FUNCTION_BLOCK PI (* PI FB *)
  (* Standard: 61499-2 *)
  (* Version 1.0, 2026-04-19, Thomas Mayr *)
  PACKAGE eclipse4diac::controlengineering;
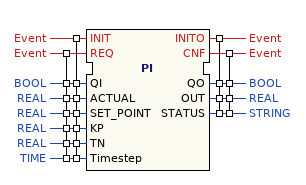
  EVENT_INPUT
    INIT WITH QI, ACTUAL, SET_POINT, KP, TN, Timestep; (* Initialize controller *)
    REQ WITH QI, ACTUAL, SET_POINT, KP, TN, Timestep; (* Execute control step *)
  END_EVENT
  EVENT_OUTPUT
    INITO WITH QO, OUT, STATUS; (* Initialization done *)
    CNF WITH QO, OUT, STATUS; (* Calculation done *)
  END_EVENT
  VAR_INPUT
    QI : BOOL; (* Enable input *)
    ACTUAL : REAL; (* Process value *)
    SET_POINT : REAL; (* Setpoint *)
    KP : REAL; (* Proportional gain *)
    TN : REAL; (* Integral time [s] *)
    Timestep : TIME; (* Sampling time (cycle time) *)
  END_VAR
  VAR_OUTPUT
    QO : BOOL; (* Enable output *)
    OUT : REAL; (* Controller output (0..100%) *)
    STATUS : STRING; (* Service Status *)
  END_VAR
  VAR
    ERR : REAL;
    I_SUM : REAL;
    DT_SEC : REAL;
  END_VAR
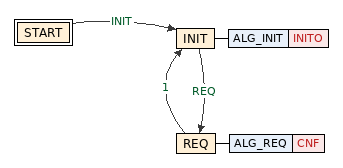
  EC_STATES
    START; (* Initial State *)
    INIT : ALG_INIT -> INITO;
    REQ : ALG_REQ -> CNF;
  END_STATES
  EC_TRANSITIONS
    START TO INIT := INIT;
    INIT TO REQ := REQ;
    REQ TO INIT := 1;
  END_TRANSITIONS
  ALGORITHM ALG_INIT IN ST:
QO := QI;
ERR := 0.0;
I_SUM := 0.0;
DT_SEC := 0.0;
OUT := 0.0;
  END_ALGORITHM
  ALGORITHM ALG_REQ IN ST:
QO := QI;

IF NOT QI THEN
	OUT := 0.0;
	I_SUM := 0.0;
ELSE
	DT_SEC := LREAL_TO_REAL(TIME_IN_S_TO_LREAL(Timestep));
	IF DT_SEC <= 0.0 OR KP <= 0.0 THEN
		STATUS := 'Inputs out of Range';
		OUT := 0.0;
	ELSE
		STATUS := 'PI Active';
		ERR := SET_POINT - ACTUAL;
		IF TN > 0.0 THEN
			IF NOT ((OUT >= 100.0 AND ERR > 0.0) OR (OUT <= 0.0 AND ERR < 0.0)) THEN
				I_SUM := I_SUM + (KP * ERR * DT_SEC / TN);
			END_IF;
		ELSE
			I_SUM := 0.0;
		END_IF;

		OUT := KP * ERR + I_SUM;

		IF OUT > 100.0 THEN
			OUT := 100.0;
		ELSIF OUT < 0.0 THEN
			OUT := 0.0;
		END_IF;
	END_IF;
END_IF;
  END_ALGORITHM
END_FUNCTION_BLOCK
